TYPE ST_LineDataParCfg :
STRUCT
    SchemaVersion : UINT := 1;  // §3.8: first member
    StaleAfterMs  : UDINT;       // mirror: declared window for staying current (§3.8e(d))
END_STRUCT
END_TYPE

(* stored: Version 1.1.0.1, ProductVersion 3.1.4024.12
   DUT ST_LineDataParCfg: Id {62645e0e-0bef-43f0-82b4-fc596d9fb9f7} *)
